FUNCTION TryConvert_REAL_TO_BOOL : BOOL
VAR_INPUT
	in : REAL;
	out : REFERENCE TO BOOL;
END_VAR

out := REAL_TO_BOOL(in);
TryConvert_REAL_TO_BOOL := TRUE;

END_FUNCTION

(* stored: Version 1.1.0.1, ProductVersion 3.1.4024.12
   POU TryConvert_REAL_TO_BOOL: Id {404ab3c5-0597-4dee-9d9b-3cfa72342579}, SpecialFunc None *)
